// This interface defines the behaviour of an interval timer, a type of timing source
// that operates based on a specified interval. It is intended to be used for periodic
// actions or repeated timing events.
INTERFACE I_IntervalTimer EXTENDS I_TimingSource

// The elapsed time since the timer was started or last reset, showing how much time has passed within the current interval.
// [get] Returns the elapsed time within the current interval.
PROPERTY ElapsedTime  : LTIME
GET
END_GET
END_PROPERTY

// The number of intervals that have elapsed since the timer was started or reset.
// [get] Returns the number of elapsed intervals.
PROPERTY IntervalCount : FsCommon.T_Size
GET
END_GET
END_PROPERTY

// The interval duration for the timer. It specifies how long the timer should wait between triggers.
// [get] Returns the interval duration.
// [set] Sets the interval duration.
PROPERTY IntervalTime : LTIME
GET
END_GET
SET
END_SET
END_PROPERTY

// Indicates whether the interval timer is currently running.
// [get] Returns TRUE if the timer is running; otherwise, FALSE.
PROPERTY IsRunning  : BOOL
GET
END_GET
END_PROPERTY

// The method that must be called cyclically to run the interval timer.
METHOD Run : I_IntervalTimer // Reference to the current instance of I_IntervalTimer.
VAR_INPUT
END_VAR
END_METHOD

// Sets the callback to be invoked when the interval has elapsed.
METHOD SetCallback : I_IntervalTimer // Reference to the current instance of I_IntervalTimer.
VAR_INPUT
	// The callback that is invoked when the interval elapses.
    ipCallback : I_TimeElapsedCallback;
END_VAR
END_METHOD

// Starts the interval timer, beginning the measurement of time intervals.
METHOD Start : I_IntervalTimer // Reference to the current instance of I_IntervalTimer.
VAR_INPUT
END_VAR
END_METHOD

// Stops the interval timer, halting the measurement of time intervals.
METHOD Stop : I_IntervalTimer // Reference to the current instance of I_IntervalTimer.
VAR_INPUT
END_VAR
END_METHOD

END_INTERFACE

(* stored: Version 1.1.0.1
   Itf I_IntervalTimer: Id {225e1e93-0d50-42d8-9923-63aeb6ddd29e}
   Property ElapsedTime: Id {739424e1-597d-4142-9976-49732fe91099}
   Get Get: Id {c39bc036-d15d-42b1-8048-7dd977fd9e99}
   Property IntervalCount: Id {69ff8348-9553-4d96-ba53-a592903a90f7}
   Get Get: Id {e35f7527-8fbb-4252-a6d6-86f668eae93d}
   Property IntervalTime: Id {69ec4c85-ca85-4387-baa5-8bc7c2e420ec}
   Get Get: Id {a74e80c7-809d-4988-bf72-4fdfce2b7f59}
   Set Set: Id {da4cf8f3-c8f6-442a-9229-ea589bf18058}
   Property IsRunning: Id {2ef0371a-ee12-4beb-90f3-869f43a48373}
   Get Get: Id {af8d5866-1674-47e0-aecc-5ab2a8d064c0}
   Method Run: Id {2c6c1dac-7cdf-4c79-9c6c-07bc8e1e2033}
   Method SetCallback: Id {48a86fe7-4282-4b9b-9db1-7871b5a00756}
   Method Start: Id {51fe5fa4-0c22-42ad-8b58-7c3b89105dd5}
   Method Stop: Id {d089fd6a-3c79-4d4c-9637-6151976ba636} *)
